TYPE StatsFault:
STRUCT
	TimeStamp: TimeStamp;
	StationID: DINT;
	FaultID: DINT;
	AcknowledgeTime: LREAL;
	Duration: LREAL;
	Data: ARRAY [0..2] OF REAL;
	StringData: ARRAY [0..3] OF STRING;
END_STRUCT
END_TYPE

(* stored: Version 1.1.0.1, ProductVersion 3.1.4024.9
   DUT StatsFault: Id {005e5626-087e-42a6-93ee-2ce986c2a8b8} *)
